FUNCTION_BLOCK FB_SEVCON
VAR_INPUT
	SEVCON_IN 		: ST_SEVCON_IN;
	Enable			: BOOL;
	ErrorReset		: BOOL;
	TargetVelocity	: UDINT;
	Self			: INT;
END_VAR
VAR_OUTPUT
	SEVCON_OUT : ST_SEVCON_OUT;
	Error		: BOOL;
	ErrorCode	: INT;
	Ready		: BOOL;
	Running		: BOOL;
END_VAR
VAR
	State		: (DEFAULT, INIT, SWITCH_ON_DISABLED, READY_TO_SWITCH_ON, SWITCHED_ON, OPERATION_ENABLED, ERROR);
	PrevState 	: (DEFAULT, INIT, SWITCH_ON_DISABLED, READY_TO_SWITCH_ON, SWITCHED_ON, OPERATION_ENABLED, ERROR);
	TimeInState	: TIME;
	StateEntry 	: BOOL;
	SwitchOn	: BOOL;
	SDO_Write		: FB_SDO_WRITE;
	SDO_WriteData	: ARRAY[0..255] OF BYTE;
	SDO_Read		: FB_SDO_READ;
	SDO_ReadData	: ARRAY[0..255] OF BYTE;
	PreChargeTimer	: TON;
	PreChargeDelay	: TIME := T#3S;
	PreChargeActive	: BOOL;
	
	HiSpeedKp		: BYTE;
	HiSpeedKi		: BYTE;
	LoSpeedKp		: BYTE;
	LoSpeedKi		: BYTE;
END_VAR
VAR CONSTANT
	VoltageMult		: REAL := 0.0625;	// Multiply by voltage params for actual voltages
	MinCapVoltage	: REAL := 40.0;		// check w/ Cedric
END_VAR



IF State <> PrevState THEN
	StateEntry := TRUE;
	PrevState := State;
ELSE
	StateEntry := FALSE;
END_IF

CASE State OF
	DEFAULT:
		State := INIT;
		
	INIT:
		// Set initial parameters
		
		Ready := FALSE;
		SEVCON_OUT.ControlWord := SevConControlWord.DisableVoltage;
		PreChargeTimer.PT := PreChargeDelay;
		
		State := SWITCH_ON_DISABLED;
		
		
	SWITCH_ON_DISABLED:
		IF StateEntry THEN
			SEVCON_OUT.ControlWord := SevConControlWord.DisableVoltage;
			SEVCON_OUT.TargetVelocity := 0;
			SEVCON_OUT.ContactorOutput := 0;
			SEVCON_OUT.BrakeOutput := 0;
		END_IF
		
		IF (SEVCON_IN.StatusWord AND SevConStatusWord.SwitchOnDisabled) = SevConStatusWord.SwitchOnDisabled THEN
			SEVCON_OUT.ControlWord := SevConControlWord.Shutdown;
			State := READY_TO_SWITCH_ON;
		END_IF
		
	READY_TO_SWITCH_ON:
		IF StateEntry THEN
			IF (SEVCON_IN.CapacitorVoltage * VoltageMult) < MinCapVoltage THEN
				PreCharge(TRUE);
			END_IF
			PreChargeTimer.IN := TRUE;
		END_IF
		
		IF ((SEVCON_IN.CapacitorVoltage * VoltageMult) > MinCapVoltage) AND PreChargeTimer.Q THEN
			SEVCON_OUT.ContactorOutput := 65535;
			PreCharge(FALSE);
			SwitchOn := TRUE;
			PreChargeTimer.IN := FALSE;
		END_IF
		
		IF SwitchOn AND ((SEVCON_IN.StatusWord AND SevConStatusWord.ReadyToSwitchon) = SevConStatusWord.ReadyToSwitchon) THEN
			SEVCON_OUT.ControlWord := SevConControlWord.SwitchOn;
			State := SWITCHED_ON;
		END_IF
	
	SWITCHED_ON:
		IF StateEntry THEN
			//
		END_IF
		
		IF (SEVCON_IN.StatusWord AND SevConStatusWord.Switchedon) = SevConStatusWord.Switchedon THEN
			Ready := TRUE;
		ELSE
			Ready := FALSE;
		END_IF
		
		IF Enable AND Ready THEN
			SEVCON_OUT.ControlWord := SevConControlWord.EnableOperation;
			State := OPERATION_ENABLED;
		END_IF

	OPERATION_ENABLED:
		IF StateEntry THEN
			SEVCON_OUT.BrakeOutput := 65535;
			Running := TRUE;
		END_IF
		
		IF NOT Enable THEN
			Running := FALSE;
			SEVCON_OUT.TargetVelocity := 0;
			IF SEVCON_IN.ActualVelocity = 0 THEN
				SEVCON_OUT.BrakeOutput := 0;
				SEVCON_OUT.ControlWord := SevConControlWord.DisableOperation;
				State := SWITCHED_ON;
			END_IF
		ELSE
			SEVCON_OUT.TargetVelocity := TargetVelocity;
		END_IF
	
	ERROR:
		IF StateEntry THEN
			Ready := FALSE;
			Error := TRUE;
		END_IF
		
		IF ErrorReset THEN
			SEVCON_OUT.ControlWord := SevConControlWord.FaultReset;
			IF (SEVCON_IN.StatusWord AND SevConStatusWord.Fault) = 0 THEN
				Error := FALSE;
				ErrorReset := FALSE;
				State := SWITCH_ON_DISABLED;
			END_IF
		END_IF
END_CASE

IF (SEVCON_IN.StatusWord AND SevConStatusWord.Fault) = SevConStatusWord.Fault THEN
	State := ERROR;
END_IF

PreChargeTimer();

METHOD PreCharge : BOOL
VAR_INPUT
	Start	: BOOL;
END_VAR
IF Start THEN
	SDO_WriteData[0] := 16#1;
	PreChargeActive := TRUE;
ELSIF NOT Start THEN
	SDO_WriteData[0] := 16#0;
	PreChargeActive := FALSE;
END_IF

SDO_WRITE(ADSNetID := '5.117.40.235.3.1',
		PortNr := CONFIG.SevCon_Port[self-1],
		CO_Index := INDEX.PreChargeActivate,
		CO_SubIndex := 0,
		DataLength := 1,
		StartWriting := TRUE,
		WriteData := SDO_WriteData);
END_METHOD

METHOD WriteTuningValues : BOOL
VAR_INPUT
	KpHi	: BYTE;
	KiHi	: BYTE;
	KpLo	: BYTE;
	KiLo	: BYTE;
END_VAR
END_METHOD

END_FUNCTION_BLOCK

(* stored: Version 1.1.0.1, ProductVersion 3.1.4024.12
   POU FB_SEVCON: Id {fa8afbbe-0b03-4d05-b50b-1bef3d1e5672}, SpecialFunc None
   Method PreCharge: Id {9fae63e7-38c4-497a-94a0-fc720c1b8126}
   Method WriteTuningValues: Id {88024c27-4d5f-4cf4-8dd4-05097a24b55a} *)
